INTERFACE I_Navitrol_DifferentialDriveMotorControl EXTENDS I_Base

{attribute 'monitoring' := 'call'}
PROPERTY EncoderCountWheelLeft : UDINT
SET
END_SET
END_PROPERTY

{attribute 'monitoring' := 'call'}
PROPERTY EncoderCountWheelRight : UDINT
SET
END_SET
END_PROPERTY

{attribute 'monitoring' := 'call'}
PROPERTY SetPointSpeedLeft : REAL
GET
END_GET
END_PROPERTY

{attribute 'monitoring' := 'call'}
PROPERTY SetPointSpeedRight : REAL
GET
END_GET
END_PROPERTY

END_INTERFACE

(* stored: Version 1.1.0.1
   Itf I_Navitrol_DifferentialDriveMotorControl: Id {97616823-74e5-495a-83c2-13fac271ce1f}
   Property EncoderCountWheelLeft: Id {1fcf0bed-4046-42af-8921-756eadccb392}
   Set Set: Id {d69b0908-2b0d-4753-9181-949b64d22321}
   Property EncoderCountWheelRight: Id {12a9c58c-d9bb-446b-bff5-fd4cf5a3ec9c}
   Set Set: Id {f424712b-9be8-452a-b47a-204498c9a71c}
   Property SetPointSpeedLeft: Id {29035341-e30a-4fe8-899a-12d6762aec54}
   Get Get: Id {758616dd-80f3-4952-94c5-ae8ad7d3bf57}
   Property SetPointSpeedRight: Id {0439bb2d-2c01-41aa-8355-9c9995d9df87}
   Get Get: Id {ac6de7f1-b155-456f-8b2c-df7b7b7bfdab} *)
